# EPICS StreamDevice protocol: protocols/mgt400.proto
Terminator = LF;
ExtraInput = Ignore;

# dma_stat_desc_push
# reply: count flags
# 62 0

# fails .. descr too long..
getFifo {
	out "\$1";
	in "%d %(\$2)d";
}

getFifoStatus {
	out "\$1";
	in "%*d %d";
}

getAuroraLaneUp {
	out "aurora_lane_up";
	in "%d";
}

getAuroraErr {
	out "aurora_errors";
	in "%d";
}
